(* IEC 61131-3 sources: RL_MAR/experiments/comparison/autoplc/results/qwen3.5-9b_20260511_180311/med_31, 1 file *)

(* ---- med_31_1.st ---- *)
FUNCTION_BLOCK ChargingStationControl
VAR_INPUT
    EVConnected : BOOL;
    EVVoltage : REAL;
    EVCurrent : REAL;
    EVStateOfCharge : REAL;
    ChargingTimer : TIME;
END_VAR
VAR_OUTPUT
    EVCharging : BOOL;
END_VAR
VAR
    VoltageOK : BOOL;
    CurrentOK : BOOL;
    SOCNotFull : BOOL;
    TimerOK : BOOL;
END_VAR

VoltageOK := (EVVoltage > 350.0);
CurrentOK := (EVCurrent <= 32.0);
SOCNotFull := (EVStateOfCharge < 100.0);
TimerOK := (ChargingTimer <= T#2h);

IF (EVConnected = TRUE) AND VoltageOK AND CurrentOK AND SOCNotFull AND TimerOK THEN
    EVCharging := TRUE;
ELSE
    EVCharging := FALSE;
END_IF;

END_FUNCTION_BLOCK
